FUNCTION_BLOCK FB_Machine EXTENDS FB_PackML_BaseModule
VAR
	Boiler		: 	I_Boiler;
	Dispenser	: I_Dispenser;
END_VAR

{warning 'Add method implementation '}
METHOD ChangeMode
VAR_INPUT
	Mode	: SPT_BaseTypes.E_PMLUnitMode;
END_VAR
END_METHOD

{warning 'Add method implementation '}
METHOD ChangeState
VAR_INPUT
	State	: SPT_BaseTypes.E_PMLCommand;
END_VAR
END_METHOD

{error 'Add property implementation or delete property to use base implementation'}
PROPERTY CurrentAlarmSeverity : SPT_BaseTypes.TcEventSeverity
GET
END_GET
END_PROPERTY

{error 'Add property implementation or delete property to use base implementation'}
PROPERTY CurrentMode : SPT_BaseTypes.E_PMLUnitMode
GET
END_GET
END_PROPERTY

{error 'Add property implementation or delete property to use base implementation'}
PROPERTY CurrentState : SPT_BaseTypes.E_PMLState
GET
END_GET
END_PROPERTY

{warning 'Add method implementation '}
METHOD CyclicLogic
END_METHOD

END_FUNCTION_BLOCK

(* stored: Version 1.1.0.1
   POU FB_Machine: Id {66cd1380-c52f-4694-bc09-18455997d862}, SpecialFunc None
   Method ChangeMode: Id {81631c5e-4939-4f96-953e-e99c88d32cc0}
   Method ChangeState: Id {3f2c94fe-6c79-416a-a6c7-76843a7ae105}
   Property CurrentAlarmSeverity: Id {50a9afe9-81c4-44b2-a8e4-9ee4e186868b}
   Get Get: Id {b77bc0c9-b905-4db6-a6bd-2875e0bb70d3}
   Property CurrentMode: Id {cdc43974-b2dd-4265-96c0-b77fd9af99ef}
   Get Get: Id {9d2df6d4-e94a-470f-95a6-8bbff4845c6c}
   Property CurrentState: Id {ee32b35c-82a9-42f2-8d73-c7ac43561ac3}
   Get Get: Id {37204a56-1ddc-4e75-80e6-f15180b608db}
   Method CyclicLogic: Id {041eac44-05ea-481d-bf59-fdcc1dd5374b} *)
